{attribute 'qualified_only'}
{attribute 'strict'}
{attribute 'to_string'}
TYPE ET_ResultShiftRegister :
(
	NotInitialised,
	LengthInvalid,
	PositionIsWrong,
	InitDone,
	RegNumberInvalid,
	GetDone,
	PutDone,
	ErrorQuitDone,
	RegisterIsEmpty,
	RegisterISFull,
	OverwriteDone,
	ReadRegisterDone
	
);
END_TYPE

(* stored: Version 1.1.0.1
   DUT ET_ResultShiftRegister: Id {f151389d-9dcc-4d99-9d9b-eafa9597b50a} *)
